// Mitsubishi GX Works2 project: PLC공장   PLC: Q03UDV

PROGRAM MAIN
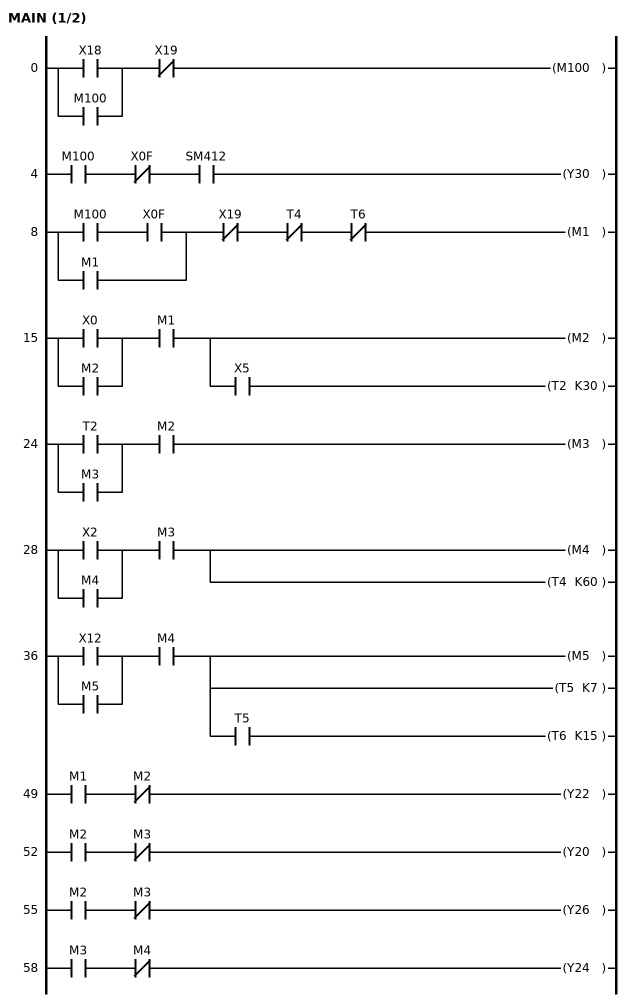
0     LD      X18
      OR      M100
      ANI     X19
      OUT     M100
4     LD      M100
      ANI     X0F
      AND     SM412
      OUT     Y30
8     LD      M100
      AND     X0F
      OR      M1
      ANI     X19
      ANI     T4
      ANI     T6
      OUT     M1
15    LD      X0
      OR      M2
      AND     M1
      OUT     M2
      AND     X5
      OUT     T2 K30
24    LD      T2
      OR      M3
      AND     M2
      OUT     M3
28    LD      X2
      OR      M4
      AND     M3
      OUT     M4
      OUT     T4 K60
36    LD      X12
      OR      M5
      AND     M4
      OUT     M5
      OUT     T5 K7
      AND     T5
      OUT     T6 K15
49    LD      M1
      ANI     M2
      OUT     Y22
52    LD      M2
      ANI     M3
      OUT     Y20
55    LD      M2
      ANI     M3
      OUT     Y26
58    LD      M3
      ANI     M4
      OUT     Y24
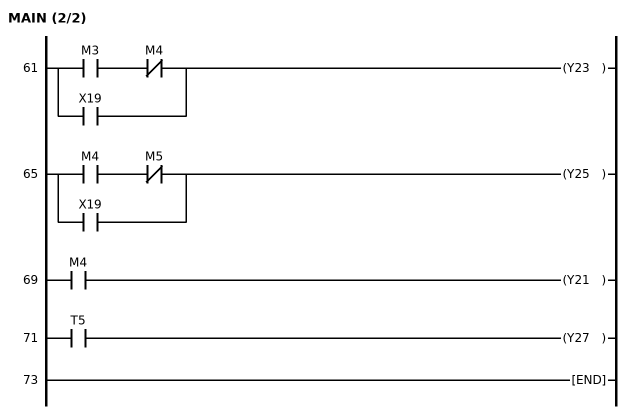
61    LD      M3
      ANI     M4
      OR      X19
      OUT     Y23
65    LD      M4
      ANI     M5
      OR      X19
      OUT     Y25
69    LD      M4
      OUT     Y21
71    LD      T5
      OUT     Y27
73    END
END_PROGRAM
